// TIA Portal V16 export
// export: Created 2021-11-12T13:32:54.7626865Z, ExportSetting WithDefaults, DisplayName Totally Integrated Automation Portal, DisplayVersion V16 Update 3, DisplayName TIA Portal Version Control Interface, DisplayVersion V16 Update 2, DisplayName TIA Portal Openness, DisplayVersion V16 Update 3, DisplayName SINAMICS Startdrive Advanced, DisplayVersion V16 Update 5, DisplayName SINAMICS Startdrive G130, G150, S120, S150, SINAMICS MV, S210, DisplayVersion V16 Update 5, DisplayName SINAMICS Startdrive G110M, G120, G120C, G120D, G120P, G115D, DisplayVersion V16 Update 5, DisplayName STEP 7 Professional, DisplayVersion V16 Update 3, DisplayName STEP 7 Safety, DisplayVersion V16, DisplayName WinCC UA Professional, DisplayVersion V16 Update 3
DATA_BLOCK "HMI_CMD_320"   // DB68
{ S7_Optimized_Access := 'TRUE' }
VERSION : 0.1
// stored: AutoNumber true, DBAccessibleFromOPCUA true, IsOnlyStoredInLoadMemory false, IsRetainMemResEnabled false, IsWriteProtectedInAS false, MemoryReserve 100
   VAR
      xxxxx___BinarySensors___xxxxx : Byte;
      "GL01-BG01" : "UDT_CH_DI_Command";   // Indukční snímač - Snímání kroku dopravníku
      "UC21-FC01_14" : "UDT_CH_DI_Command";   // 400V Dopravník ++320 (K1) OK
      xxxxx___BinaryOthers___xxxxx : Byte;
      SF02_14 : "UDT_CH_DI_Command";   // Conveyor Remote / Dopravník Remote
      SF02_24 : "UDT_CH_DI_Command";   // Conveyor Automat / Dopravník Automat
      SF03_14 : "UDT_CH_DI_Command";   // Conveyor Manual Backward / Dopravník Manuál Vzad
      SF03_24 : "UDT_CH_DI_Command";   // Conveyor Manual Forward / Dopravník Manual Vpřed
      SF04_14 : "UDT_CH_DI_Command";   // Conveyor Start automat / Dopravník Start automat
      SF05_12 : "UDT_CH_DI_Command";   // Conveyor Stop / Dopravník Stop
      xxxxx___Drives___xxxxx : Byte;
      "GL01-MA01" : "UDT_Drive1_Command";   // Pohon dopravníku - Dopravník z kalicí vany (K1)
      "UC21-TA01" : "UDT_SINAMICS_G120_Command";   // Měnič
      xxxxx__Alarms__xxxxx : Byte;
      "GL01-MA01_1" : "UDT_DI_Mon_Command";   // v daném čase nedosažena pozice - taktovací mód
   END_VAR
BEGIN
END_DATA_BLOCK
